Fanuc KAREL source: w_multi.kl

PROGRAM w_multi
%NOLOCKGROUP
VAR
  p : POSITION
  q : POSITION
  i : INTEGER
  r : REAL
BEGIN
  WITH $SPEED = r, $MOTYPE = i, $TERMTYPE = NODECEL MOVE TO p
  WITH $SPEED = 200 MOVE TO q NOWAIT
  WITH $SPEED = 100 MOVE NEAR p BY 50.0
END w_multi
